{attribute 'GeneratedUsingTerminal: EK1100-0000-0018'}
{attribute addProperty BoxType "EK1100-0000-0018"}
{attribute addProperty Id "Term_10_EK1122Term_10_EK1122_BB9FBBE4214Term_23_EL3403EL3403_812980A665Term_24_EL6001EL6001_0DE01E7E61Term_25_EL3024EL3024_C6E76B5A40Term_19_EL9011EL9011_D65D3D320"}
{attribute addProperty CRC "2014708462"}
{attribute addProperty Size "380"}
TYPE Term_9_EK1100_781602EE EXTENDS EK1100_1FC0878B :
STRUCT
	{attribute addProperty Name "Term 10 (EK1122)"}
	{attribute addProperty PreviousPort "Term 9 (EK1100) : B"}
	Term_10_EK1122 : Term_10_EK1122_BB9FBBE4;
	{attribute addProperty Name "Term 23 (EL3403)"}
	{attribute addProperty PreviousPort "Term 10 (EK1122) : C"}
	Term_23_EL3403 : EL3403_812980A6;
	{attribute addProperty Name "Term 24 (EL6001)"}
	{attribute addProperty PreviousPort "Term 23 (EL3403) : B"}
	Term_24_EL6001 : EL6001_0DE01E7E;
	{attribute addProperty Name "Term 25 (EL3024)"}
	{attribute addProperty PreviousPort "Term 24 (EL6001) : B"}
	Term_25_EL3024 : EL3024_C6E76B5A;
	{attribute addProperty Name "Term 19 (EL9011)"}
	{attribute addProperty PreviousPort "Term 25 (EL3024) : B"}
	Term_19_EL9011 : EL9011_D65D3D32;
END_STRUCT
END_TYPE

(* stored: Version 1.2.0.0, ProductVersion 3.1.4024.9
   DUT Term_9_EK1100_781602EE: Id {57d03584-d2b0-0e0b-0c8e-687aa27ec655} *)
